FUNCTION f_DelBit64 : LWORD
VAR_INPUT
  inVal   : LWORD;
  bitNo   : INT;
END_VAR
VAR
  wConst : LWORD := 1;
END_VAR

IF ( inVal AND SHL( wConst,INT_TO_SINT(bitNo) MOD 64 ) ) > 0 THEN
  f_DelBit64 := inVal XOR (SHL( wConst,INT_TO_SINT(bitNo) MOD 64 ));
ELSE
  f_DelBit64 := inVal;
END_IF

END_FUNCTION

(* stored: Version 1.1.0.1, ProductVersion 3.1.4022.18
   POU f_DelBit64: Id {40002ec8-591e-429b-87fd-872ad82375c0}, SpecialFunc None *)
